FUNCTION_BLOCK FB_EventBuffer

VAR
MemRingBuffer: FB_MemRingBuffer;	
aBufferArray  : ARRAY[0..Number_Of_Bytes_For_All_ST_Event] OF BYTE; (* Buffer memory used by FB_MemRingBuffer function block *)
END_VAR

VAR CONSTANT
	Size_Of_ST_Event: UDINT :=SIZEOF(ST_Event);
	Max_Number_Of_ST_Event: UDINT := 5;
	Number_Of_Bytes_For_All_ST_Event: UDINT := Size_Of_ST_Event*Max_Number_Of_ST_Event;
END_VAR

METHOD PUBLIC GetAndRemoveEvent
VAR_OUTPUT
	stEvent: ST_Event;
	bError : BOOL;
END_VAR
MemRingBuffer.A_RemoveHead(pRead:=ADR(stEvent),
						  	cbRead:=SIZEOF(stEvent),
							pBuffer:=ADR(aBufferArray),
							cbBuffer:=SIZEOF(aBufferArray));

bError:= NOT MemRingBuffer.bOk;
END_METHOD

METHOD PUBLIC TryToAddEvent
VAR_INPUT
	stEvent: REFERENCE TO ST_Event;
END_VAR

VAR_OUTPUT
    bError : BOOL;
END_VAR
MemRingBuffer.A_AddTail(pWrite:=ADR(stEvent),
						cbWrite:=SIZEOF(stEvent),
						pBuffer:=ADR(aBufferArray),cbBuffer:=SIZEOF(aBufferArray));
bError:= NOT MemRingBuffer.bOk;
END_METHOD

END_FUNCTION_BLOCK

(* stored: Version 1.1.0.1, ProductVersion 3.1.4024.12
   POU FB_EventBuffer: Id {086ae6cc-a776-4b87-9805-b5c83d0ad2e4}, SpecialFunc None
   Method GetAndRemoveEvent: Id {542fcee9-c4d9-439b-b25d-8b85f18f933e}
   Method TryToAddEvent: Id {5a363483-42f2-4186-8867-7c5405833674} *)
